FUNCTION_BLOCK SUBL_1 (* 2-variable data subscriber *)
  (* Standard: 61499-2 *)
  (* Version 1.0, 21-03-12, GASR, Universidade do Estado de Santa Catarina *)
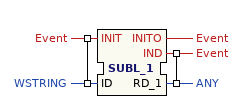
  EVENT_INPUT
    INIT WITH ID; (* Service initiaization *)
  END_EVENT
  EVENT_OUTPUT
    INITO; (* Initialization confirm *)
    IND WITH RD_1; (* Service indication *)
  END_EVENT
  VAR_INPUT
    ID : WSTRING; (* Default id is the FB instance name *)
  END_VAR
  VAR_OUTPUT
    RD_1 : ANY;
  END_VAR
END_FUNCTION_BLOCK
